FUNCTION_BLOCK ButtonConsole
  (* Standard: 61499-2 *)
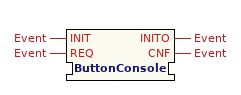
  EVENT_INPUT
    INIT;
    REQ;
  END_EVENT
  EVENT_OUTPUT
    INITO;
    CNF;
  END_EVENT
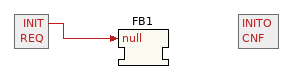
  FBS
    FB1 : ;
  END_FBS
  EVENT_CONNECTIONS
    INIT TO FB1.null;
  END_CONNECTIONS
END_FUNCTION_BLOCK
